TYPE stLimit  :
STRUCT
    rMinimumValue : REAL;      // Lower bound for the REAL value to be tested 
    rMaxiumValue : REAL;      // Upper bound for the REAL value to be tested 
    bValueMustBe : BOOL;      // Whtere if the varirable BOOL must be TRUE or FALSE
END_STRUCT
END_TYPE

(* stored: Version 1.1.0.1, ProductVersion 3.1.4024.16
   DUT stLimit: Id {d07cec05-3e96-43b8-ae05-922e9211aeaf} *)
